Staubli VAL3: showExist.pgx

program showExist(string x_sName, string x_sMessage)
  local string l_sMessage
  local string l_sMessage2
begin
  // not possibile to delete rename
  call language:message(l_sMessage,23)
  call language:message(l_sMessage2,29)
  l_sMessage=l_sMessage+x_sName
  popUpMsg(l_sMessage+l_sMessage2+x_sMessage)
end
